Staubli VAL3: clkPark2.pgx

program clkPark2()
begin
  // -- move back to initial position
  resetMotion()
  movej(jInitialPosition,tTool,mNomSpeed)
  waitEndMove()
end
